// TIA Portal project "NUEVA PRACTICA MEJORADA CARGA DESCARGA" (V17)

(* hardware
DEVICE "Estación S7-1500/ET200MP_1"  S7-1500 station
   slot 0: "Perfil soporte_0"  Rack  6ES7 590-1***0-0AA0
   slot 1: "PLC_1"  CPU 1513-1 PN  6ES7 513-1AL01-0AB0  V2.9
      slot 3: "Display de la CPU_1"  6ES7591-1AA00-0AA0
      slot 32768: "Interfaz PROFINET_1"  X1
         slot 32769: "Puerto_1"  X1 P1
         slot 32770: "Puerto_2"  X1 P2
      slot 34817: "Virtual CP interface port_1"  Virtual CP interface port  Virtual CP interface port
   slot 2: "AI 8xU/I/RTD/TC ST_1"  AI 8xU/I/RTD/TC ST  6ES7 531-7KF00-0AB0  V2.0
   slot 3: "AI 8xU/I/RTD/TC ST_2"  AI 8xU/I/RTD/TC ST  6ES7 531-7KF00-0AB0  V2.0
   slot 4: "AI 8xU/I/RTD/TC ST_3"  AI 8xU/I/RTD/TC ST  6ES7 531-7KF00-0AB0  V2.0
   slot 5: "AI 8xU/I/RTD/TC ST_4"  AI 8xU/I/RTD/TC ST  6ES7 531-7KF00-0AB0  V2.0
   slot 6: "DI 16x24VDC BA_1"  DI 16x24VDC BA  6ES7 521-1BH10-0AA0  V1.0
*)

// ===== PLC "PLC_1"  CPU 1513-1 PN =====

VAR_GLOBAL   // PLC tag table "Tabla de variables estándar"
   "Start" AT %I20.0 : Bool;
   "Stop" AT %I20.1 : Bool;
   "1At Entry" AT %I20.2 : Bool;
   "1At Load" AT %I20.3 : Bool;
   "1At Left" AT %I20.4 : Bool;
   "1At Right" AT %I20.5 : Bool;
   "1At Middle" AT %I20.6 : Bool;
   "1Moving x" AT %I20.7 : Bool;
   "1Moving Z" AT %I21.0 : Bool;
   "2At Exit" AT %I21.1 : Bool;
   "2At Unload" AT %I21.2 : Bool;
   "2Left Limit" AT %I21.3 : Bool;
   "2Stacker Crane o Right Limit" AT %I21.4 : Bool;
   "2Middle Limit" AT %I21.5 : Bool;
   "2 Moving-X" AT %I21.6 : Bool;
   "2Moving-Z" AT %I21.7 : Bool;
   "Reset" AT %I22.0 : Bool;
   "Start light" AT %Q20.0 : Bool;
   "1Emitter" AT %Q20.1 : Bool;
   "1Entry Conveyor" AT %Q20.2 : Bool;
   "1Load Conveyor" AT %Q20.3 : Bool;
   "1Forks Left" AT %Q20.4 : Bool;
   "1Forks Right" AT %Q20.5 : Bool;
   "1Lift" AT %Q20.6 : Bool;
   "2Remover" AT %Q20.7 : Bool;
   "2Exit Conveyor" AT %Q21.0 : Bool;
   "2load Conveyor" AT %Q21.1 : Bool;
   "2Stacker Left" AT %Q21.2 : Bool;
   "2Stacker Right" AT %Q21.3 : Bool;
   "2Lift" AT %Q21.4 : Bool;
   "suma1" AT %QW30 : Int;
   "suma2" AT %QW32 : Int;
   "CAJA MG" AT %QW34 : Int;
   "motor1" AT %Q21.5 : Bool;
   "PISTON 1" AT %Q21.6 : Bool;
   "RECEPTOR MG" AT %I22.1 : Bool;
   "Pusher 0" AT %I22.2 : Bool;
   "START1" AT %I22.3 : Bool;
   "START1 LIGHT" AT %Q21.7 : Bool;
   "MANUAL" AT %I22.4 : Bool;
   "STACK LIGHT" AT %Q22.0 : Bool;
   "STACK LIGHT1" AT %Q22.1 : Bool;
   "1Target Position" AT %QW36 : Int;
   "2Target Position" AT %QW38 : Int;
   "x" AT %I22.5 : Bool;
   "contador1" AT %I22.6 : Bool;
   "contador2" AT %I22.7 : Bool;
END_VAR

DATA_BLOCK "EMITTER_DB"   // DB1
{ S7_Optimized_Access := 'TRUE' }
VERSION : 0.1
// stored: InstanceOfName EMITTER
"EMITTER"
BEGIN
END_DATA_BLOCK

DATA_BLOCK "ALMACCEN_DB"   // DB4
{ S7_Optimized_Access := 'TRUE' }
VERSION : 0.1
// stored: InstanceOfName ALMACCEN
"ALMACCEN"
BEGIN
   CUENTA2 := 0;
END_DATA_BLOCK

// folder: System blocks/Program resources

DATA_BLOCK "contador 2"   // DB2
{ S7_Optimized_Access := 'TRUE' }
AUTHOR : Simatic
FAMILY : IEC
NAME : CNTR
VERSION : 1.0
// stored: InstanceOfName IEC_COUNTER
"IEC_COUNTER"
BEGIN
END_DATA_BLOCK

DATA_BLOCK "CI_DB"   // DB3
{ S7_Optimized_Access := 'TRUE' }
AUTHOR : Simatic
FAMILY : IEC
NAME : CNTR
VERSION : 1.0
// stored: InstanceOfName IEC_COUNTER
"IEC_COUNTER"
BEGIN
END_DATA_BLOCK

DATA_BLOCK "IEC_Counter_0_DB"   // DB5
{ S7_Optimized_Access := 'TRUE' }
AUTHOR : Simatic
FAMILY : IEC
NAME : CNTR
VERSION : 1.0
// stored: InstanceOfName IEC_COUNTER
"IEC_COUNTER"
BEGIN
END_DATA_BLOCK

DATA_BLOCK "IEC_Timer_0_DB"   // DB6
{ S7_Optimized_Access := 'TRUE' }
AUTHOR : Simatic
FAMILY : IEC
NAME : IEC_TMR
VERSION : 1.0
// stored: InstanceOfName IEC_TIMER
"IEC_TIMER"
BEGIN
END_DATA_BLOCK

DATA_BLOCK "contador1v1"   // DB7
{ S7_Optimized_Access := 'TRUE' }
AUTHOR : Simatic
FAMILY : IEC
NAME : CNTR
VERSION : 1.0
// stored: InstanceOfName IEC_COUNTER
"IEC_COUNTER"
BEGIN
END_DATA_BLOCK

DATA_BLOCK "contador2v2"   // DB8
{ S7_Optimized_Access := 'TRUE' }
AUTHOR : Simatic
FAMILY : IEC
NAME : CNTR
VERSION : 1.0
// stored: InstanceOfName IEC_COUNTER
"IEC_COUNTER"
BEGIN
END_DATA_BLOCK

// folder: (top level)

FUNCTION_BLOCK "ALMACCEN"   // FB1, LAD
TITLE = *** CARGA DESCARGA DE LAS ESTANTERIAS DE UNA NAVE***
{ S7_Optimized_Access := 'TRUE' }
VERSION : 0.1
   VAR_INPUT
      Start : Bool;
      MANUAL : Bool;
      start1 : Bool;
      Stop : Bool;
      "1At Entry" : Bool;
      "1At Load" : Bool;
      "1At Left" : Bool;
      "1At Right" : Bool;
      "1At Middle" : Bool;
      "1Moving x" : Bool;
      "1Moving Z" : Bool;
      "2At Exit" : Bool;
      "2At Unload" : Bool;
      "2Left Limit" : Bool;
      "2Stacker Crane o Right Limit" : Bool;
      "2Middle Limit" : Bool;
      "2 Moving-X" : Bool;
      "2Moving-Z" : Bool;
      Reset : Bool;
   END_VAR
   VAR_OUTPUT
      "STACK LIGHT1" : Bool;
      "STACK LIGHT" : Bool;
      "Start light" : Bool;
      "STAR1 LIGHT" : Bool;
      "1Emitter" : Bool;
      "1Entry Conveyor" : Bool;
      "1Load Conveyor" : Bool;
      "1Forks Left" : Bool;
      "1Forks Right" : Bool;
      "1Lift" : Bool;
      "2Remover" : Bool;
      "2Exit Conveyor" : Bool;
      "2load Conveyor" : Bool;
      "2Stacker Left" : Bool;
      "2Stacker Right" : Bool;
      "1Targe Position" : Int;
      "2Targe Position" : Int;
      "2Lift" : Bool;
   END_VAR
   VAR
      CUENTA1 : Int;
      CUENTA2 : Int := 1;
      K : Bool;
      K1 : Bool;
      "X1 AT LOAD(1)" : Bool;
      "AUX0(1)" : Bool;
      "AUX1(1)" : Bool;
      "AUX2(1)" : Bool;
      "AUX3(1)" : Bool;
      "AUX4(1)" : Bool;
      "AUXCONT(1)" : Bool;
      "X(1)" : Bool;
      "X0(1)" : Bool;
      "X1(1)" : Bool;
      "X2(1)" : Bool;
      "X3(1)" : Bool;
      "X4(1)" : Bool;
      "XF(1)" : Bool;
      "X1 AT EXIT(2)" : Bool;
      "AUX0(2)" : Bool;
      "AUX1(2)" : Bool;
      "AUX2(2)" : Bool;
      "AUX3(2)" : Bool;
      "AUX4(2)" : Bool;
      "AUXCONT(2)" : Bool;
      "X(2)" : Bool;
      "X0(2)" : Bool;
      "X1(2)" : Bool;
      "X2(2)" : Bool;
      "X3(2)" : Bool;
      "X4(2)" : Bool;
      "X5(2)" : Bool;
      "XF(2)" : Bool;
      CUENTA_TOPE : Int := 54;
      FLANCO0 : Bool;
      FLANCO1 : Bool;
      FLANCO2 : Bool;
      FLANCO3 : Bool;
      FLANCO4 : Bool;
      FLANCO6 : Bool;
      FLANCO5 : Bool;
      FLANCO7 : Bool;
      FLANCO8 : Bool;
      FLANCO9 : Bool;
      FLANCO10 : Bool;
      FLANCO11 : Bool;
      FLANCO12 : Bool;
      FLANCO13 : Bool;
      FLANCO14 : Bool;
      FLANCO15 : Bool;
      FLANCO16 : Bool;
      FLANCO17 : Bool;
      FLANCO18 : Bool;
      FLANCO19 : Bool;
      FLANCO20 : Bool;
      FLANCO21 : Bool;
      FLANCO22 : Bool;
      FLANCO23 : Bool;
      "T1-1" : TON_TIME;
      "T2-1" : TON_TIME;
      "T3-1" : TON_TIME;
      T4 : TON_TIME;
      T5 : TON_TIME;
      T6 : TON_TIME;
      T7 : TON_TIME;
      T8 : TON_TIME;
      T9 : TON_TIME;
      T10 : TON_TIME;
      T11 : TON_TIME;
      T12 : TON_TIME;
      retardo : TON_TIME;
   END_VAR
   VAR_TEMP   // added for the SCL form of the ladder/FBD networks
      _w1 : Bool;
      _w2 : Bool;
      _w3 : Bool;
      _w4 : Bool;
      _w5 : Bool;
      _w6 : Bool;
      _w7 : Bool;
      _w8 : Bool;
      _w9 : Bool;
      _w10 : Bool;
      _w11 : Bool;
   END_VAR
BEGIN

REGION Network 1: ***MOVIMIENTO DEL PRIMER APILADOR***
   // identificados todos los movimientos activamos cintas y las posiciones del primer apilador.
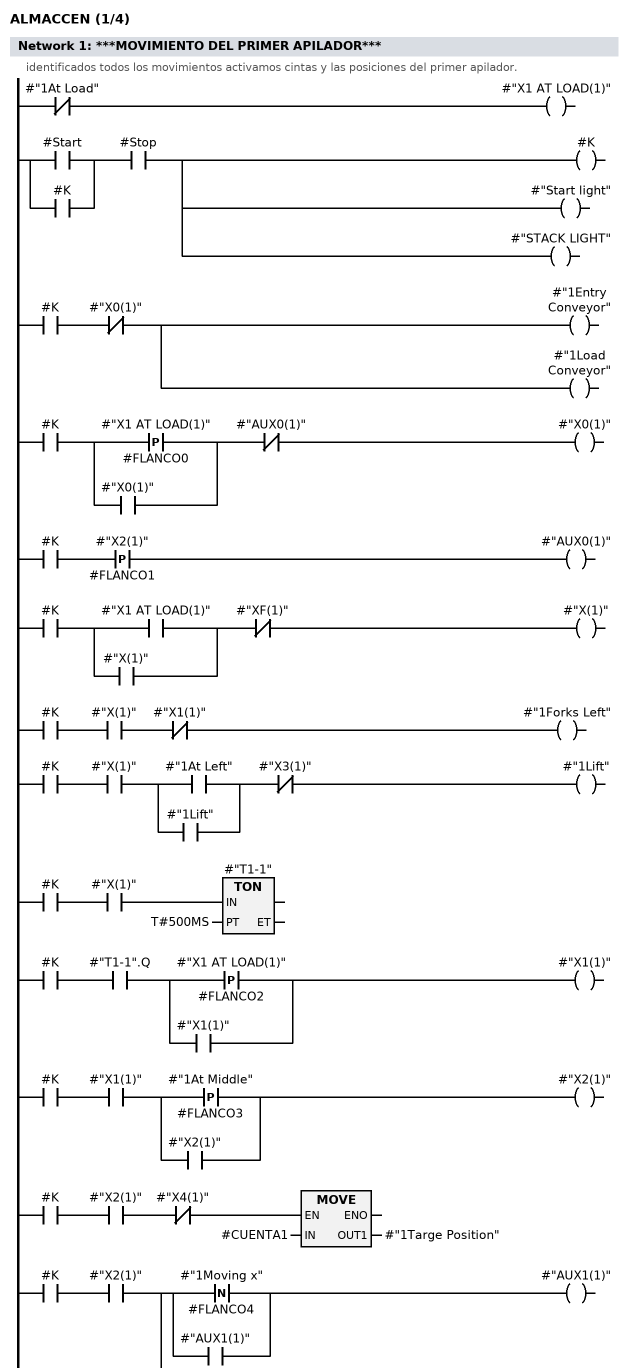
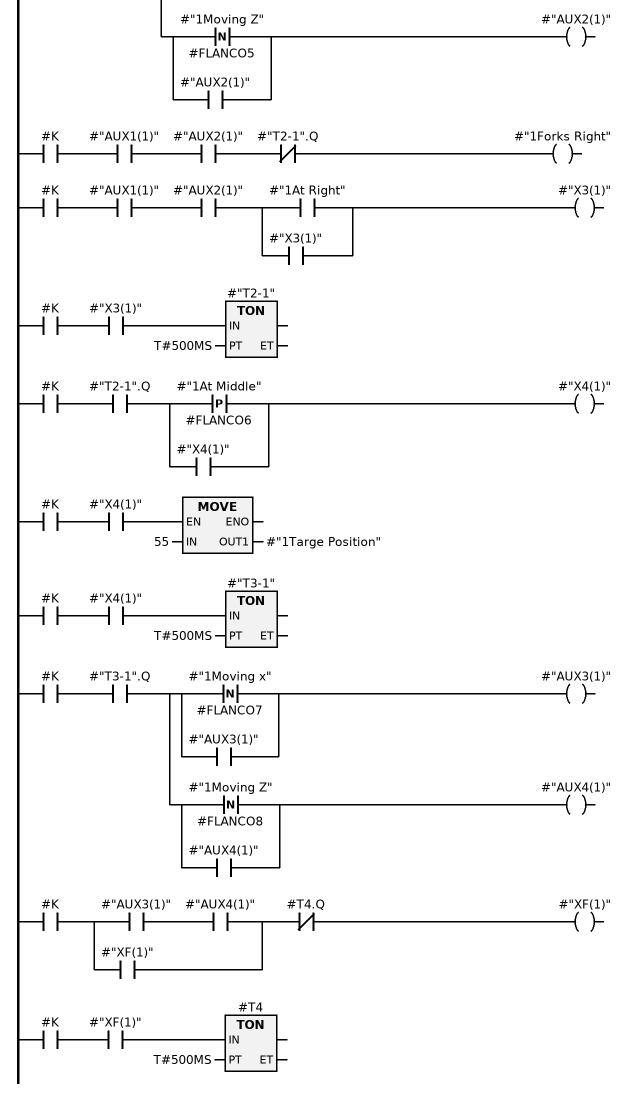
   #"X1 AT LOAD(1)" := NOT #"1At Load";
   #K := (#Start OR #K) AND #Stop;
   #"Start light" := #K;
   #"STACK LIGHT" := #K;
   #"1Entry Conveyor" := #K AND NOT #"X0(1)";
   #"1Load Conveyor" := #"1Entry Conveyor";
   #_w1 := #K AND #"X1 AT LOAD(1)" AND NOT #FLANCO0;   // rising edge of #"X1 AT LOAD(1)"
   #FLANCO0 := #"X1 AT LOAD(1)";
   #"X0(1)" := (#_w1 OR (#K AND #"X0(1)")) AND NOT #"AUX0(1)";
   #_w2 := #K AND #"X2(1)" AND NOT #FLANCO1;   // rising edge of #"X2(1)"
   #FLANCO1 := #"X2(1)";
   #"AUX0(1)" := #_w2;
   #"X(1)" := #K AND (#"X1 AT LOAD(1)" OR #"X(1)") AND NOT #"XF(1)";
   #"1Forks Left" := #K AND #"X(1)" AND NOT #"X1(1)";
   #"1Lift" := #K AND #"X(1)" AND (#"1At Left" OR #"1Lift") AND NOT #"X3(1)";
   #"T1-1"(IN := #K AND #"X(1)", PT := T#500MS);   // TON
   #_w3 := #K AND #"T1-1".Q AND #"X1 AT LOAD(1)" AND NOT #FLANCO2;   // rising edge of #"X1 AT LOAD(1)"
   #FLANCO2 := #"X1 AT LOAD(1)";
   #"X1(1)" := #_w3 OR (#K AND #"T1-1".Q AND #"X1(1)");
   #_w4 := #K AND #"X1(1)" AND #"1At Middle" AND NOT #FLANCO3;   // rising edge of #"1At Middle"
   #FLANCO3 := #"1At Middle";
   #"X2(1)" := #_w4 OR (#K AND #"X1(1)" AND #"X2(1)");
   IF #K AND #"X2(1)" AND NOT #"X4(1)" THEN #"1Targe Position" := #CUENTA1; END_IF;
   #_w5 := #K AND #"X2(1)";
   #_w6 := #_w5 AND NOT #"1Moving x" AND #FLANCO4;   // falling edge of #"1Moving x"
   #FLANCO4 := #"1Moving x";
   #"AUX1(1)" := #_w6 OR (#_w5 AND #"AUX1(1)");
   #_w7 := #_w5 AND NOT #"1Moving Z" AND #FLANCO5;   // falling edge of #"1Moving Z"
   #FLANCO5 := #"1Moving Z";
   #"AUX2(1)" := #_w7 OR (#_w5 AND #"AUX2(1)");
   #"1Forks Right" := #K AND #"AUX1(1)" AND #"AUX2(1)" AND NOT #"T2-1".Q;
   #"X3(1)" := #K AND #"AUX1(1)" AND #"AUX2(1)" AND (#"1At Right" OR #"X3(1)");
   #"T2-1"(IN := #K AND #"X3(1)", PT := T#500MS);   // TON
   #_w8 := #K AND #"T2-1".Q AND #"1At Middle" AND NOT #FLANCO6;   // rising edge of #"1At Middle"
   #FLANCO6 := #"1At Middle";
   #"X4(1)" := #_w8 OR (#K AND #"T2-1".Q AND #"X4(1)");
   IF #K AND #"X4(1)" THEN #"1Targe Position" := 55; END_IF;
   #"T3-1"(IN := #K AND #"X4(1)", PT := T#500MS);   // TON
   #_w9 := #K AND #"T3-1".Q;
   #_w10 := #_w9 AND NOT #"1Moving x" AND #FLANCO7;   // falling edge of #"1Moving x"
   #FLANCO7 := #"1Moving x";
   #"AUX3(1)" := #_w10 OR (#_w9 AND #"AUX3(1)");
   #_w11 := #_w9 AND NOT #"1Moving Z" AND #FLANCO8;   // falling edge of #"1Moving Z"
   #FLANCO8 := #"1Moving Z";
   #"AUX4(1)" := #_w11 OR (#_w9 AND #"AUX4(1)");
   #"XF(1)" := #K AND ((#"AUX3(1)" AND #"AUX4(1)") OR #"XF(1)") AND NOT #T4.Q;
   #T4(IN := #K AND #"XF(1)", PT := T#500MS);   // TON
END_REGION

REGION Network 2: *** CONTADOR DEL PRIMER APILADOR ESTE EN CONSTANTE FUNCIONAMIENTO***
   // Contador del primer carrito para saber su posicion y pulsador para que siempre este funcionando y no haya ningun 0 en el contador, por que lee de 1 a 54.
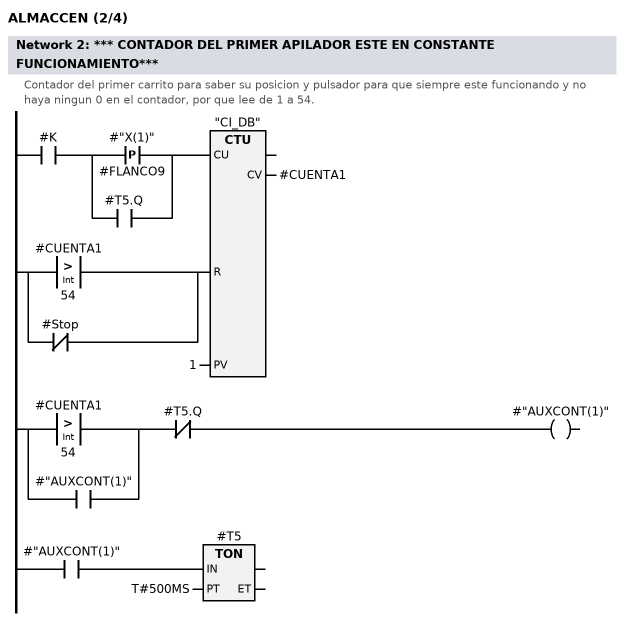
   #_w1 := #K AND #"X(1)" AND NOT #FLANCO9;   // rising edge of #"X(1)"
   #FLANCO9 := #"X(1)";
   "CI_DB".CTU(CU := #_w1 OR (#K AND #T5.Q), R := (#CUENTA1 > 54) OR NOT #Stop, PV := 1, CV => #CUENTA1);
   #"AUXCONT(1)" := ((#CUENTA1 > 54) OR #"AUXCONT(1)") AND NOT #T5.Q;
   #T5(IN := #"AUXCONT(1)", PT := T#500MS);   // TON
END_REGION

REGION Network 3: ++++AUTOMATICO++++++
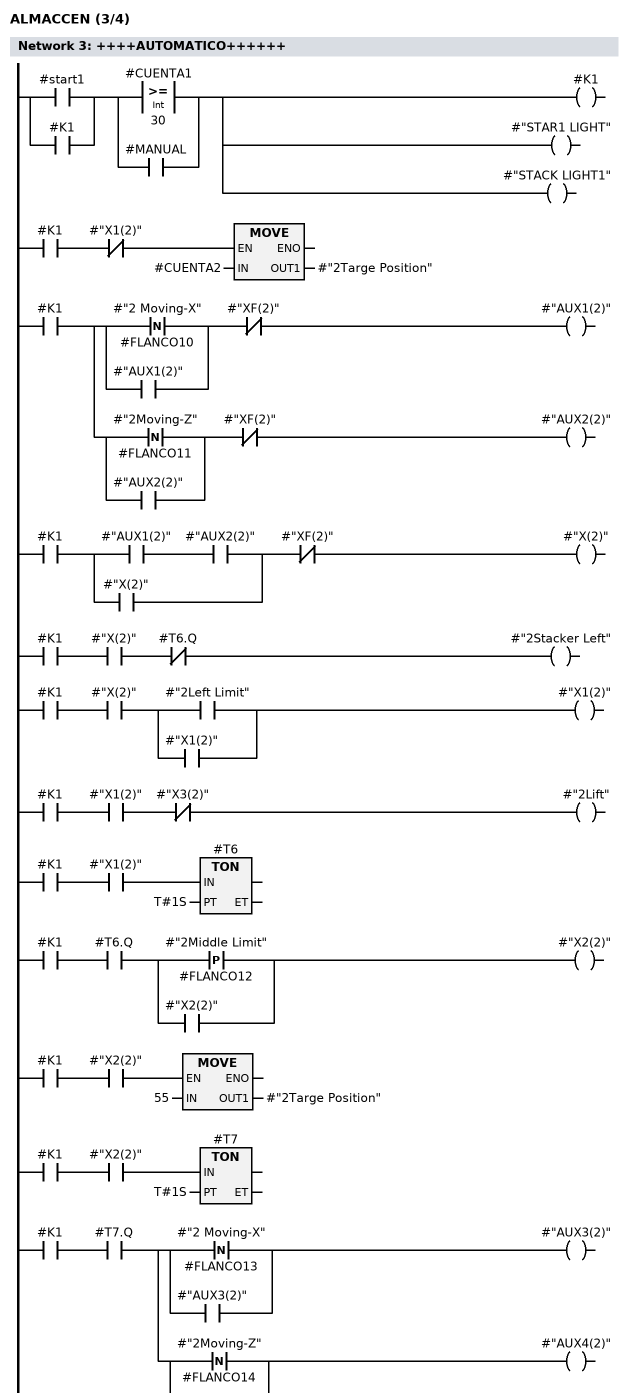
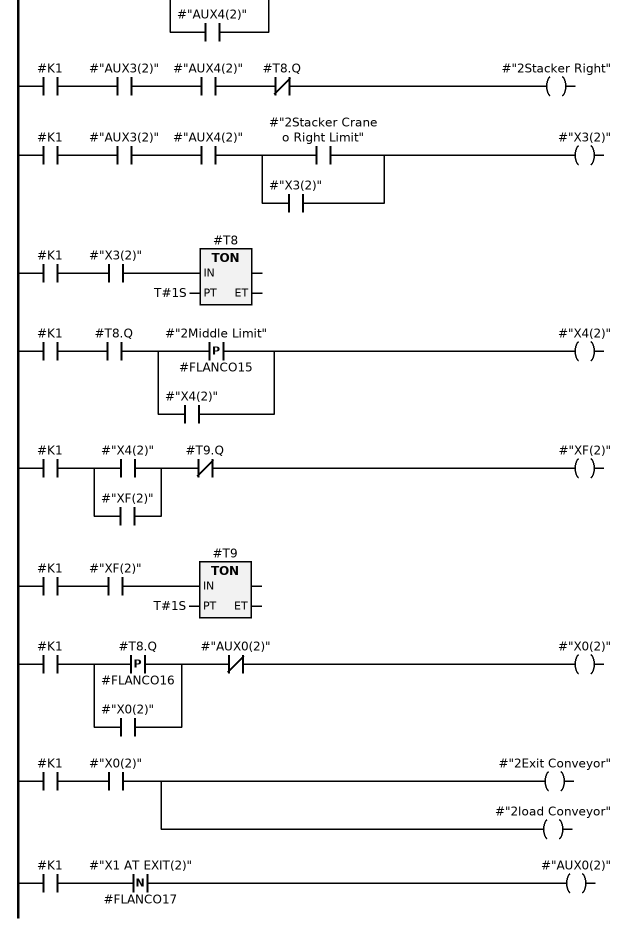
   #K1 := (#start1 OR #K1) AND ((#CUENTA1 >= 30) OR #MANUAL);
   #"STAR1 LIGHT" := #K1;
   #"STACK LIGHT1" := #K1;
   IF #K1 AND NOT #"X1(2)" THEN #"2Targe Position" := #CUENTA2; END_IF;
   #_w1 := #K1 AND NOT #"2 Moving-X" AND #FLANCO10;   // falling edge of #"2 Moving-X"
   #FLANCO10 := #"2 Moving-X";
   #"AUX1(2)" := (#_w1 OR (#K1 AND #"AUX1(2)")) AND NOT #"XF(2)";
   #_w2 := #K1 AND NOT #"2Moving-Z" AND #FLANCO11;   // falling edge of #"2Moving-Z"
   #FLANCO11 := #"2Moving-Z";
   #"AUX2(2)" := (#_w2 OR (#K1 AND #"AUX2(2)")) AND NOT #"XF(2)";
   #"X(2)" := #K1 AND ((#"AUX1(2)" AND #"AUX2(2)") OR #"X(2)") AND NOT #"XF(2)";
   #"2Stacker Left" := #K1 AND #"X(2)" AND NOT #T6.Q;
   #"X1(2)" := #K1 AND #"X(2)" AND (#"2Left Limit" OR #"X1(2)");
   #"2Lift" := #K1 AND #"X1(2)" AND NOT #"X3(2)";
   #T6(IN := #K1 AND #"X1(2)", PT := T#1S);   // TON
   #_w3 := #K1 AND #T6.Q AND #"2Middle Limit" AND NOT #FLANCO12;   // rising edge of #"2Middle Limit"
   #FLANCO12 := #"2Middle Limit";
   #"X2(2)" := #_w3 OR (#K1 AND #T6.Q AND #"X2(2)");
   IF #K1 AND #"X2(2)" THEN #"2Targe Position" := 55; END_IF;
   #T7(IN := #K1 AND #"X2(2)", PT := T#1S);   // TON
   #_w4 := #K1 AND #T7.Q;
   #_w5 := #_w4 AND NOT #"2 Moving-X" AND #FLANCO13;   // falling edge of #"2 Moving-X"
   #FLANCO13 := #"2 Moving-X";
   #"AUX3(2)" := #_w5 OR (#_w4 AND #"AUX3(2)");
   #_w6 := #_w4 AND NOT #"2Moving-Z" AND #FLANCO14;   // falling edge of #"2Moving-Z"
   #FLANCO14 := #"2Moving-Z";
   #"AUX4(2)" := #_w6 OR (#_w4 AND #"AUX4(2)");
   #"2Stacker Right" := #K1 AND #"AUX3(2)" AND #"AUX4(2)" AND NOT #T8.Q;
   #"X3(2)" := #K1 AND #"AUX3(2)" AND #"AUX4(2)" AND (#"2Stacker Crane o Right Limit" OR #"X3(2)");
   #T8(IN := #K1 AND #"X3(2)", PT := T#1S);   // TON
   #_w7 := #K1 AND #T8.Q AND #"2Middle Limit" AND NOT #FLANCO15;   // rising edge of #"2Middle Limit"
   #FLANCO15 := #"2Middle Limit";
   #"X4(2)" := #_w7 OR (#K1 AND #T8.Q AND #"X4(2)");
   #"XF(2)" := #K1 AND (#"X4(2)" OR #"XF(2)") AND NOT #T9.Q;
   #T9(IN := #K1 AND #"XF(2)", PT := T#1S);   // TON
   #_w8 := #K1 AND #T8.Q AND NOT #FLANCO16;   // rising edge of #T8.Q
   #FLANCO16 := #T8.Q;
   #"X0(2)" := (#_w8 OR (#K1 AND #"X0(2)")) AND NOT #"AUX0(2)";
   #"2Exit Conveyor" := #K1 AND #"X0(2)";
   #"2load Conveyor" := #"2Exit Conveyor";
   #_w9 := #K1 AND NOT #"X1 AT EXIT(2)" AND #FLANCO17;   // falling edge of #"X1 AT EXIT(2)"
   #FLANCO17 := #"X1 AT EXIT(2)";
   #"AUX0(2)" := #_w9;
END_REGION

REGION Network 4: *** CONTADOR SEGUNDO APILADOR ***
   // Igual manera que el primer contador para activar y descativar
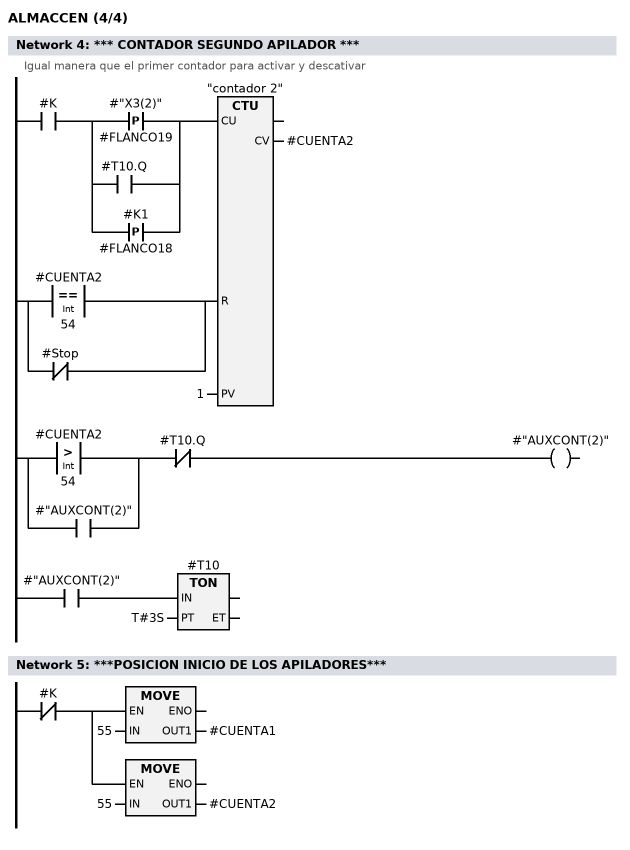
   #_w1 := #K AND #"X3(2)" AND NOT #FLANCO19;   // rising edge of #"X3(2)"
   #FLANCO19 := #"X3(2)";
   #_w2 := #K AND #K1 AND NOT #FLANCO18;   // rising edge of #K1
   #FLANCO18 := #K1;
   "contador 2".CTU(CU := #_w1 OR (#K AND #T10.Q) OR #_w2,
                    R := (#CUENTA2 = 54) OR NOT #Stop,
                    PV := 1,
                    CV => #CUENTA2);
   #"AUXCONT(2)" := ((#CUENTA2 > 54) OR #"AUXCONT(2)") AND NOT #T10.Q;
   #T10(IN := #"AUXCONT(2)", PT := T#3S);   // TON
END_REGION

REGION Network 5: ***POSICION INICIO DE LOS APILADORES***
   RUNG wire#powerrail
      I_Contact( #K )
      wire#w1
      Move(in := 55, out1 => #CUENTA1)
   END_RUNG
   RUNG wire#w1
      Move(in := 55, out1 => #CUENTA2)
   END_RUNG
   // the same network as SCL:
   IF NOT #K THEN
       #CUENTA1 := 55;
       #CUENTA2 := 55;
   END_IF;
END_REGION
END_FUNCTION_BLOCK

FUNCTION_BLOCK "EMITTER"   // FB2, LAD
{ S7_Optimized_Access := 'TRUE' }
VERSION : 0.1
// EMITER PARA QUE SIEMPRE SALGAN CAJAS,ESTE RETARDO SE PUDE COFIGURAR EN FACTORYIO
   VAR_INPUT
      K : Bool;
      SENSOR : Bool;
      Pusher : Bool;
   END_VAR
   VAR_OUTPUT
      EMITTER : Bool;
   END_VAR
   VAR
      EMITTER1 : Bool;
      EMITTER2 : Bool;
      EMITER3 : Bool;
      T1 : TON_TIME;
      T2 : TON_TIME;
      T3 : TON_TIME;
   END_VAR
BEGIN

REGION Network 1: *** EMITTER***
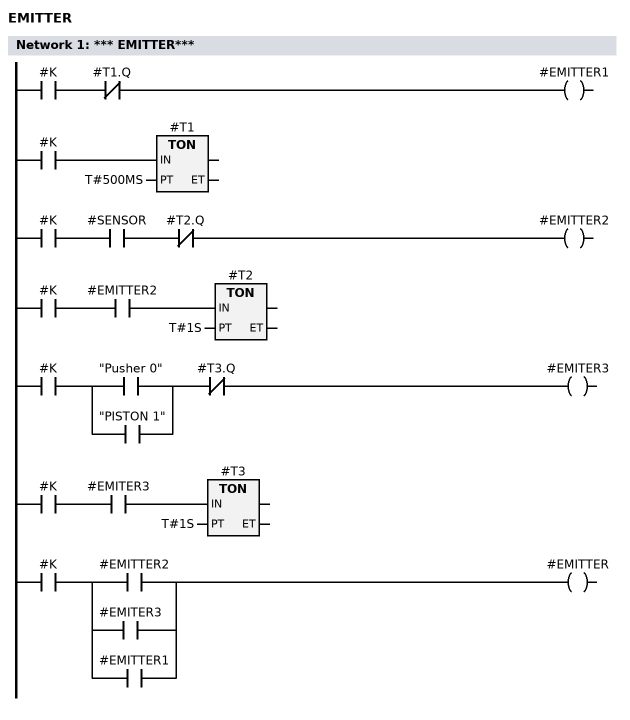
   #EMITTER1 := #K AND NOT #T1.Q;
   #T1(IN := #K, PT := T#500MS);   // TON
   #EMITTER2 := #K AND #SENSOR AND NOT #T2.Q;
   #T2(IN := #K AND #EMITTER2, PT := T#1S);   // TON
   #EMITER3 := #K AND ("Pusher 0" OR "PISTON 1") AND NOT #T3.Q;
   #T3(IN := #K AND #EMITER3, PT := T#1S);   // TON
   #EMITTER := #K AND (#EMITTER2 OR #EMITER3 OR #EMITTER1);
END_REGION
END_FUNCTION_BLOCK

FUNCTION "MHJ-PLC-Lab-Function-S71500" : Void   // FC9000, SCL
{ S7_Optimized_Access := 'TRUE' }
VERSION : 0.1
   VAR_TEMP
      Value : Byte;
      ForCounter : Int;
   END_VAR
   VAR CONSTANT
      Value_01_DW : DWord := 16#1223_5486;
      Value_02_DW : DWord := 16#A6C9_D1F5;
   END_VAR
BEGIN

   #Value:=PEEK(area := 16#82,
        dbNumber := 0,
        byteOffset := 511);
   #Value := #Value + 1;

   POKE(area := 16#82,
        dbNumber := 0,
        byteOffset := 511,
        value := #Value);

   POKE(area := 16#82,
        dbNumber := 0,
        byteOffset := 1016,
        value := #Value_01_DW);
   POKE(area := 16#82,
        dbNumber := 0,
        byteOffset := 1020,
        value := #Value_02_DW);

   FOR #ForCounter := 0 TO 63 DO
       #Value:=PEEK(area := 16#1,
            dbNumber := 0,
            byteOffset := #ForCounter);
       POKE(area := 16#81,
            dbNumber := 0,
            byteOffset := #ForCounter,
            value := #Value);
   END_FOR;
   #Value := PEEK(area := 16#1,
                  dbNumber := 0,
                  byteOffset := 512);
   POKE(area := 16#82,
        dbNumber := 0,
        byteOffset := 512,
        value := #Value);
END_FUNCTION

ORGANIZATION_BLOCK "Main"   // OB1, LAD, ProgramCycle
TITLE = "Main Program Sweep (Cycle)"
{ S7_Optimized_Access := 'TRUE' }
VERSION : 0.1
   VAR_INPUT
      Initial_Call : Bool;   // Initial call of this OB
      Remanence : Bool;   // =True, if remanent data are available
   END_VAR
   VAR_TEMP   // added for the SCL form of the ladder/FBD networks
      _w1 : Bool;
   END_VAR
BEGIN

REGION Network 1: CARRO DEPOSITA Y SUELTA
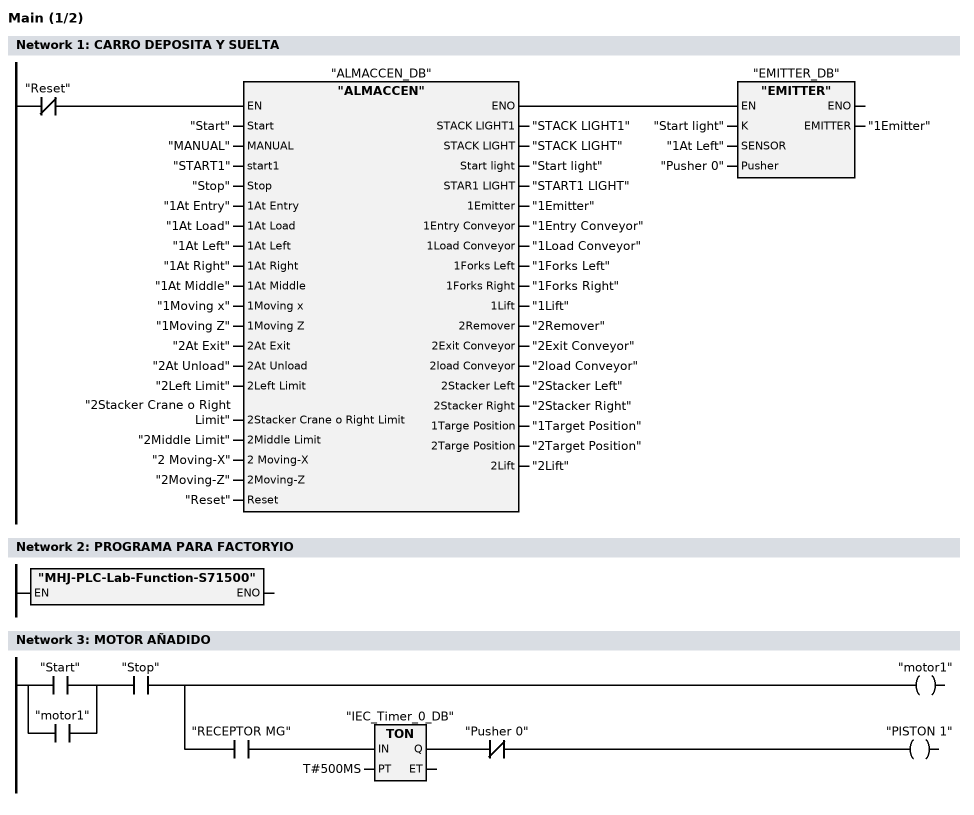
   RUNG wire#powerrail
      I_Contact( "Reset" )
      "ALMACCEN_DB"(Start := "Start", MANUAL := "MANUAL", start1 := "START1", Stop := "Stop", "1At Entry" := "1At Entry", "1At Load" := "1At Load", "1At Left" := "1At Left", "1At Right" := "1At Right", "1At Middle" := "1At Middle", "1Moving x" := "1Moving x", "1Moving Z" := "1Moving Z", "2At Exit" := "2At Exit", "2At Unload" := "2At Unload", "2Left Limit" := "2Left Limit", "2Stacker Crane o Right Limit" := "2Stacker Crane o Right Limit", "2Middle Limit" := "2Middle Limit", "2 Moving-X" := "2 Moving-X", "2Moving-Z" := "2Moving-Z", Reset := "Reset", "STACK LIGHT1" => "STACK LIGHT1", "STACK LIGHT" => "STACK LIGHT", "Start light" => "Start light", "STAR1 LIGHT" => "START1 LIGHT", "1Emitter" => "1Emitter", "1Entry Conveyor" => "1Entry Conveyor", "1Load Conveyor" => "1Load Conveyor", "1Forks Left" => "1Forks Left", "1Forks Right" => "1Forks Right", "1Lift" => "1Lift", "2Remover" => "2Remover", "2Exit Conveyor" => "2Exit Conveyor", "2load Conveyor" => "2load Conveyor", "2Stacker Left" => "2Stacker Left", "2Stacker Right" => "2Stacker Right", "1Targe Position" => "1Target Position", "2Targe Position" => "2Target Position", "2Lift" => "2Lift")
      "EMITTER_DB"(K := "Start light", SENSOR := "1At Left", Pusher := "Pusher 0", EMITTER => "1Emitter")
   END_RUNG
   // the same network as SCL:
   "ALMACCEN_DB"(EN := NOT "Reset",   // "ALMACCEN"
                 Start := "Start",
                 MANUAL := "MANUAL",
                 start1 := "START1",
                 Stop := "Stop",
                 "1At Entry" := "1At Entry",
                 "1At Load" := "1At Load",
                 "1At Left" := "1At Left",
                 "1At Right" := "1At Right",
                 "1At Middle" := "1At Middle",
                 "1Moving x" := "1Moving x",
                 "1Moving Z" := "1Moving Z",
                 "2At Exit" := "2At Exit",
                 "2At Unload" := "2At Unload",
                 "2Left Limit" := "2Left Limit",
                 "2Stacker Crane o Right Limit" := "2Stacker Crane o Right Limit",
                 "2Middle Limit" := "2Middle Limit",
                 "2 Moving-X" := "2 Moving-X",
                 "2Moving-Z" := "2Moving-Z",
                 Reset := "Reset",
                 "STACK LIGHT1" => "STACK LIGHT1",
                 "STACK LIGHT" => "STACK LIGHT",
                 "Start light" => "Start light",
                 "STAR1 LIGHT" => "START1 LIGHT",
                 "1Emitter" => "1Emitter",
                 "1Entry Conveyor" => "1Entry Conveyor",
                 "1Load Conveyor" => "1Load Conveyor",
                 "1Forks Left" => "1Forks Left",
                 "1Forks Right" => "1Forks Right",
                 "1Lift" => "1Lift",
                 "2Remover" => "2Remover",
                 "2Exit Conveyor" => "2Exit Conveyor",
                 "2load Conveyor" => "2load Conveyor",
                 "2Stacker Left" => "2Stacker Left",
                 "2Stacker Right" => "2Stacker Right",
                 "1Targe Position" => "1Target Position",
                 "2Targe Position" => "2Target Position",
                 "2Lift" => "2Lift",
                 ENO => #_w1);
   IF #_w1 THEN
       "EMITTER_DB"(K := "Start light", SENSOR := "1At Left", Pusher := "Pusher 0", EMITTER => "1Emitter");   // "EMITTER"
   END_IF;
END_REGION

REGION Network 2: PROGRAMA PARA FACTORYIO
   RUNG wire#powerrail
      "MHJ-PLC-Lab-Function-S71500"()
   END_RUNG
   // the same network as SCL:
   "MHJ-PLC-Lab-Function-S71500"();
END_REGION

REGION Network 3: MOTOR AÑADIDO
   "motor1" := ("Start" OR "motor1") AND "Stop";
   "IEC_Timer_0_DB".TON(IN := "motor1" AND "RECEPTOR MG", PT := T#500MS);
   "PISTON 1" := "IEC_Timer_0_DB".Q AND NOT "Pusher 0";
END_REGION

REGION Network 4: CONTADOR DISPLEY
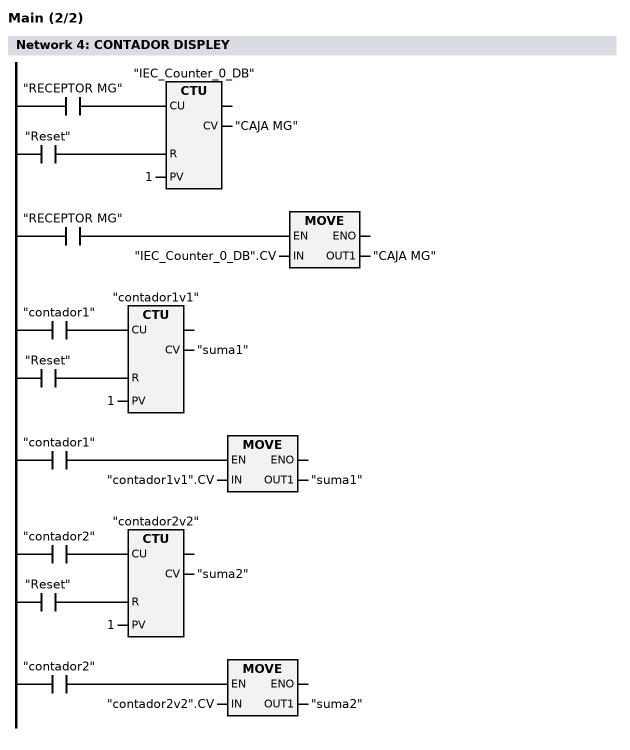
   "IEC_Counter_0_DB".CTU(CU := "RECEPTOR MG", R := "Reset", PV := 1, CV => "CAJA MG");
   IF "RECEPTOR MG" THEN "CAJA MG" := "IEC_Counter_0_DB".CV; END_IF;
   "contador1v1".CTU(CU := "contador1", R := "Reset", PV := 1, CV => "suma1");
   IF "contador1" THEN "suma1" := "contador1v1".CV; END_IF;
   "contador2v2".CTU(CU := "contador2", R := "Reset", PV := 1, CV => "suma2");
   IF "contador2" THEN "suma2" := "contador2v2".CV; END_IF;
END_REGION
END_ORGANIZATION_BLOCK